ABB RobotStudio station: w2.rspag

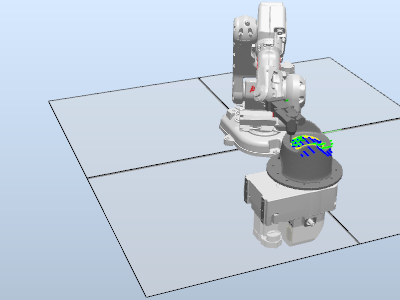
--- station ---
Station Project1 (saved by RobotStudio 22.3.10098.0)
Controller Controller1
  mechanical unit ROB_1: IRB140_6_81_C_03, 6 joints, base frame (0, 0, 0) mm
  mechanical unit M7DM1: MTD_250_M2009_REV1_01, 1 joints, base frame (684.98, -128.75, 250) mm, rotated rx 0 ry 0 rz 90 deg
Layout (positions relative to the parent item):
  - IRB140_6_81_C_03 [mechanism, from Robots\IRB140_6_81_C_G_03.rslib] at (0, 0, 0) mm; joint values [-0.4404, 0.1901, 0.3733, 2.4186, 0.7001, -2.5479] (rad or m)
  - MTD_250_M2009_REV1_01 [mechanism] at (684.98, -128.75, 250) mm, rotated rx 0 ry 0 rz 90 deg; joint values [0] (rad or m)
      links: Base, Link1
  - gripped_pen [mechanism, from MNFG309\gripped_pen.rslib] at (480.48, -195.8, 502.57) mm, rotated rx 97.75 ry 90 rz 97.75 deg
  - potty1 [part] at (798.66, 39.43, 241.77) mm, rotated rx 90 ry 0 rz 0 deg, size 275.1 x 194.8 x 257.3 mm
Attachment: gripped_pen is attached to IRB140_6_81_C_03 / Link6
Attachment: potty1 is attached to MTD_250_M2009_REV1_01 / Link1
Attachment: potty is attached to potty1
Targets, tools, work objects and paths stored in the station and not in the controller backup, written as RAPID:
! task T_ROB1
MODULE CalibData
  PERS tooldata gripped_pen:=[TRUE,[[121,0,178],[1,0,0,0]],[2,[0,50,88],[1,0,0,0],0,0,0]];
  TASK PERS wobjdata potty:=[FALSE,TRUE,"",[[684.978108354,-128.746939063,250],[0.707106781,0,0,0.707106781]],[[0,0,0],[1,0,0,0]]];
ENDMODULE

! task T_ROB1
MODULE Module1
  CONST robtarget Target_10:=[[-45.03,50.16,129.476],[0.5,0.5,0.5,-0.5],[-1,1,-2,0],[9E+09,9E+09,9E+09,9E+09,9E+09,9E+09]];
  CONST robtarget Target_20:=[[-20.282,62.744,129.127],[0.5,0.5,0.5,-0.5],[-1,1,-2,0],[9E+09,9E+09,9E+09,9E+09,9E+09,9E+09]];
  CONST robtarget Target_30:=[[11.896,64.483,128.86],[0.5,0.5,0.5,-0.5],[0,2,-3,0],[9E+09,9E+09,9E+09,9E+09,9E+09,9E+09]];
  CONST robtarget Target_40:=[[39.689,53.042,128.927],[0.5,0.5,0.5,-0.5],[0,2,-3,0],[9E+09,9E+09,9E+09,9E+09,9E+09,9E+09]];
  CONST robtarget Target_50:=[[57.798,34.115,127.1],[0.5,0.5,0.5,-0.5],[0,2,-3,0],[9E+09,9E+09,9E+09,9E+09,9E+09,9E+09]];
  CONST robtarget Target_60:=[[68.525,10.908,127.738],[0.5,0.5,0.5,-0.5],[0,2,-3,0],[9E+09,9E+09,9E+09,9E+09,9E+09,9E+09]];
  CONST robtarget Target_70:=[[70.794,-19.857,128.419],[0.5,0.5,0.5,-0.5],[0,2,-3,0],[9E+09,9E+09,9E+09,9E+09,9E+09,9E+09]];
  CONST robtarget Target_80:=[[62.436,-48.353,129.808],[0.5,0.5,0.5,-0.5],[0,2,-3,0],[9E+09,9E+09,9E+09,9E+09,9E+09,9E+09]];
  CONST robtarget Target_90:=[[45.201,-69.327,131.428],[0.5,0.5,0.5,-0.5],[0,2,-3,0],[9E+09,9E+09,9E+09,9E+09,9E+09,9E+09]];
  CONST robtarget Target_100:=[[21.201,-86.605,140.96],[0.5,0.5,0.5,-0.5],[0,2,-3,0],[9E+09,9E+09,9E+09,9E+09,9E+09,9E+09]];
  CONST robtarget Target_110:=[[-9.927,-98.657,169.887],[0.5,0.5,0.5,-0.5],[-1,1,-2,0],[9E+09,9E+09,9E+09,9E+09,9E+09,9E+09]];
  CONST robtarget Target_120:=[[-49.23,-86.236,170.954],[0.5,0.5,0.5,-0.5],[-1,1,-2,0],[9E+09,9E+09,9E+09,9E+09,9E+09,9E+09]];
  CONST robtarget Target_130:=[[-64.618,-62.853,148.116],[0.5,0.5,0.5,-0.5],[-1,1,-2,0],[9E+09,9E+09,9E+09,9E+09,9E+09,9E+09]];
  CONST robtarget Target_140:=[[-74.299,-32.791,131.037],[0.5,0.5,0.5,-0.5],[-1,1,-2,0],[9E+09,9E+09,9E+09,9E+09,9E+09,9E+09]];
  CONST robtarget Target_150:=[[-76.984,-1.82,131.395],[0.5,0.5,0.5,-0.5],[-1,1,-2,0],[9E+09,9E+09,9E+09,9E+09,9E+09,9E+09]];
  CONST robtarget Target_160:=[[-67.051,26.501,131.572],[0.5,0.5,0.5,-0.5],[-1,1,-2,0],[9E+09,9E+09,9E+09,9E+09,9E+09,9E+09]];
  PROC Path_10()
    MoveL Target_10,v1000,z100,gripped_pen\WObj:=potty;
    MoveL Target_20,v1000,z100,gripped_pen\WObj:=potty;
    MoveL Target_30,v1000,z100,gripped_pen\WObj:=potty;
    MoveL Target_40,v1000,z100,gripped_pen\WObj:=potty;
    MoveL Target_50,v1000,z100,gripped_pen\WObj:=potty;
    MoveL Target_60,v1000,z100,gripped_pen\WObj:=potty;
    MoveL Target_70,v1000,z100,gripped_pen\WObj:=potty;
    MoveL Target_80,v1000,z100,gripped_pen\WObj:=potty;
    MoveL Target_90,v1000,z100,gripped_pen\WObj:=potty;
    MoveL Target_100,v1000,z100,gripped_pen\WObj:=potty;
    MoveL Target_110,v1000,z100,gripped_pen\WObj:=potty;
    MoveL Target_120,v1000,z100,gripped_pen\WObj:=potty;
    MoveL Target_130,v1000,z100,gripped_pen\WObj:=potty;
    MoveL Target_140,v1000,z100,gripped_pen\WObj:=potty;
    MoveL Target_150,v1000,z100,gripped_pen\WObj:=potty;
    MoveL Target_160,v1000,z100,gripped_pen\WObj:=potty;
  ENDPROC
ENDMODULE


--- Controller Data/Controller1/RAPID/TASK1/PROGMOD/Module1.mod ---
MODULE Module1
    !***********************************************************
    !
    ! Module:  Module1
    !
    ! Description:
    !   <Insert description here>
    !
    ! Author: sgmxu9
    !
    ! Version: 1.0
    !
    !***********************************************************


    !***********************************************************
    !
    ! Procedure main
    !
    !   This is the entry point of your program
    !
    !***********************************************************
    PROC main()
        !Add your code here
    ENDPROC
ENDMODULE

--- Controller Data/Controller1/SYSPAR/EIO.cfg ---
EIO:CFG_1.0:6:1::
#
INDUSTRIAL_NETWORK:

      -Name "DeviceNet" -Label "DeviceNet Master/Slave Network" -Address "2"
#
DEVICENET_INTERNAL_DEVICE:

      -Name "DN_Internal_Device" -VendorName "ABB Robotics"\
      -ProductName "DeviceNet Internal Slave Device"
